// TIA Portal V17 export
// export: Created 2023-12-22T15:28:35.6842744Z, ExportSetting WithDefaults, DisplayName Totally Integrated Automation Portal, DisplayVersion V17, DisplayName TIA Portal Openness, DisplayVersion V17, DisplayName TIA Portal Version Control Interface, DisplayVersion V17, DisplayName STEP 7 Professional, DisplayVersion V17, DisplayName STEP 7 Safety, DisplayVersion V17, DisplayName WinCC Advanced, DisplayVersion V17
FUNCTION_BLOCK "DIx_1"   // FB200, LAD
{ S7_Optimized_Access := 'FALSE' }
VERSION : 0.1
// Input - входной сигнал контроллера
// pulse - частота фильтрации дребезга
// Signal - обработанный и отфильтрованный сигнал, используемый в дальнейшем
// stored: AutoNumber false, IsIECCheckEnabled false, SetENOAutomatically false, UDAEnableTagReadback false
   VAR
      AllBlock { S7_SetPoint := 'True'} : "DI_ex";   // 2.4 разрешение на работу
      signal_2 { S7_SetPoint := 'True'} : "DI_ex";   // 2.3 Нижний уровень
      signal_3 { S7_SetPoint := 'True'} : "DI_ex";   // Ротаметр 1
      signal_4 { S7_SetPoint := 'True'} : "DI_ex";   // Ротаметр 2
      signal_5 { S7_SetPoint := 'True'} : "DI_ex";   // Ротаметр 3
      signal_6 { S7_SetPoint := 'True'} : "DI_ex";   // Датчик переливва
      signal_7 { S7_SetPoint := 'True'} : "DI_ex";   // Датчик переливва
      signal_8 { S7_SetPoint := 'True'} : "DI_ex";
      signal_9 { S7_SetPoint := 'True'} : "DI_ex";
      signal_10 { S7_SetPoint := 'True'} : "DI_ex";
      signal_11 { S7_SetPoint := 'True'} : "DI_ex";
      signal_12 { S7_SetPoint := 'True'} : "DI_ex";
   END_VAR
   VAR DB_SPECIFIC
      Time_DTL { S7_SetPoint := 'True'} : DTL;
   END_VAR
   VAR_TEMP   // added for the SCL form of the ladder/FBD networks
      _w1 : Bool;
   END_VAR
BEGIN

REGION Network 1: AllBlock
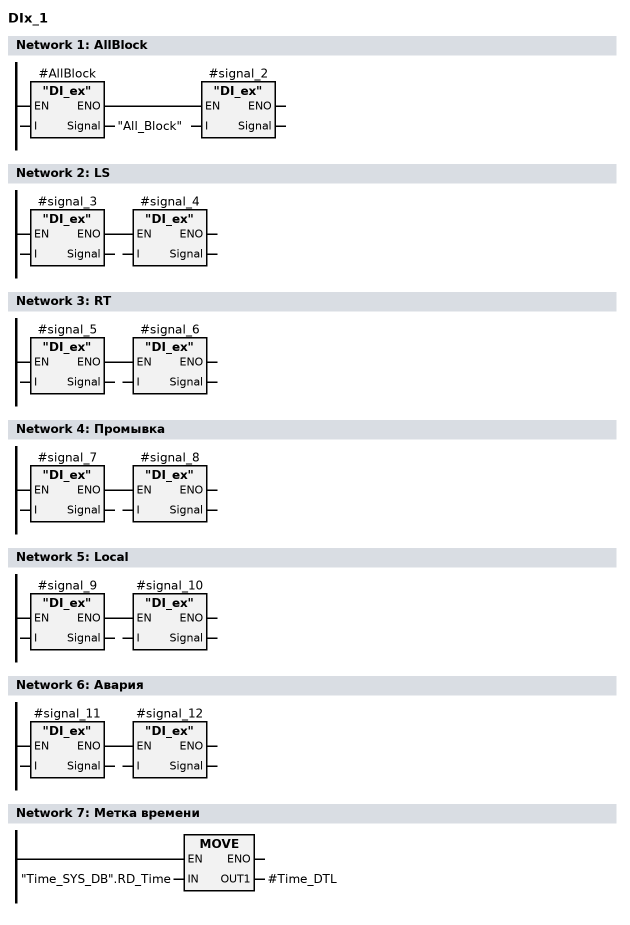
   RUNG wire#powerrail
      #AllBlock(I :=, Signal => "All_Block")
      #signal_2(I :=, Signal =>)
   END_RUNG
   // the same network as SCL:
   #AllBlock(Signal => "All_Block", ENO => #_w1);   // "DI_ex"
   IF #_w1 THEN
       #signal_2();   // "DI_ex"
   END_IF;
END_REGION

REGION Network 2: LS
   RUNG wire#powerrail
      #signal_3(I :=, Signal =>)
      #signal_4(I :=, Signal =>)
   END_RUNG
   // the same network as SCL:
   #signal_3(ENO => #_w1);   // "DI_ex"
   IF #_w1 THEN
       #signal_4();   // "DI_ex"
   END_IF;
END_REGION

REGION Network 3: RT
   RUNG wire#powerrail
      #signal_5(I :=, Signal =>)
      #signal_6(I :=, Signal =>)
   END_RUNG
   // the same network as SCL:
   #signal_5(ENO => #_w1);   // "DI_ex"
   IF #_w1 THEN
       #signal_6();   // "DI_ex"
   END_IF;
END_REGION

REGION Network 4: Промывка
   RUNG wire#powerrail
      #signal_7(I :=, Signal =>)
      #signal_8(I :=, Signal =>)
   END_RUNG
   // the same network as SCL:
   #signal_7(ENO => #_w1);   // "DI_ex"
   IF #_w1 THEN
       #signal_8();   // "DI_ex"
   END_IF;
END_REGION

REGION Network 5: Local
   RUNG wire#powerrail
      #signal_9(I :=, Signal =>)
      #signal_10(I :=, Signal =>)
   END_RUNG
   // the same network as SCL:
   #signal_9(ENO => #_w1);   // "DI_ex"
   IF #_w1 THEN
       #signal_10();   // "DI_ex"
   END_IF;
END_REGION

REGION Network 6: Авария
   RUNG wire#powerrail
      #signal_11(I :=, Signal =>)
      #signal_12(I :=, Signal =>)
   END_RUNG
   // the same network as SCL:
   #signal_11(ENO => #_w1);   // "DI_ex"
   IF #_w1 THEN
       #signal_12();   // "DI_ex"
   END_IF;
END_REGION

REGION Network 7: Метка времени
   RUNG wire#powerrail
      Move(in := "Time_SYS_DB".RD_Time, out1 => #Time_DTL)
   END_RUNG
   // the same network as SCL:
   #Time_DTL := "Time_SYS_DB".RD_Time;
END_REGION
END_FUNCTION_BLOCK
